// TwinCAT 3 PLC project SandBox
// ProgramVersion: 3.1.4026.22
// libraries:
//   [Logging Helper], * (Beckhoff Industrial)
//   Tc2_Standard, * (Beckhoff Automation GmbH)
//   Tc2_System, * (Beckhoff Automation GmbH)
// project tree:
//   / MAIN.TcPOU, PlcTask.TcTTO
//   Source/ MotionArgument.TcPOU, ST_MotionParameters.TcDUT
// (motion and I/O tree: see PLC project unittestplc)
// real-time tasks:
//   TASK PlcTask: cycle T#10ms, priority 20, ADS port 350
//   TASK PlcTask1: cycle T#10ms, priority 21, ADS port 351

CONFIGURATION SandBox
    RESOURCE PLC ON TwinCAT3
        TASK PlcTask(INTERVAL := T#10ms, PRIORITY := 21);
        PROGRAM MAIN WITH PlcTask : MAIN;
    END_RESOURCE
END_CONFIGURATION

// ---- Source/ST_MotionParameters.TcDUT
TYPE ST_MotionParameters :
	STRUCT
		Velocity : LREAL;
		Accel	 : LREAL;
		Decel	 : LREAL;
		Jerk	 : LREAL;
	END_STRUCT
END_TYPE

// ---- MAIN.TcPOU
PROGRAM MAIN
VAR
	Logger			: LogHelper<2>;
	LocalLog		: LocalLogger;
	initialized		: BOOL;
	Message			: LogMessage;
	Source			: LogSource;
	MotionArg		: MotionArgument;
	MotionParameters : ST_MotionParameters;
	
	//Commands
	logNoArgument	: BOOL;
	logWithArgument : BOOL;
END_VAR

IF NOT initialized THEN
	initialized			 := TRUE;
	MotionArg.Parameters REF= MotionParameters;
	Logger.Subscribe(LocalLog);
END_IF

IF logNoArgument THEN
	Source.SourceName := 'Test';
	Source.Timestamp := 123456789;
	Message.Message := 'Message';
	Message.Severity := 12;
	Logger.LogMessage(Source, Message);
	logNoArgument := FALSE;
END_IF

IF logWithArgument THEN
	Logger.LogMessage(Source, Message, MotionArg);
	logWithArgument := FALSE;
END_IF

END_PROGRAM

// ---- Source/MotionArgument.TcPOU
FUNCTION_BLOCK MotionArgument IMPLEMENTS I_LogArgument
VAR
	_Pars : REFERENCE TO ST_MotionParameters;
END_VAR

PROPERTY Parameters : REFERENCE TO ST_MotionParameters
GET
Parameters := _Pars;
END_GET
SET
_Pars REF= Parameters;
END_SET
END_PROPERTY

METHOD ToString : Logging_Helper.T_MaxString
ToString := CONCAT('Vel: ', CONCAT(TO_STRING(_Pars.Velocity), CONCAT(' Accel: ', CONCAT(TO_STRING(_Pars.Accel), CONCAT(' Decel: ', CONCAT(TO_STRING(_Pars.Decel), CONCAT(' Jerk: ',TO_STRING(_Pars.Jerk))))))));
END_METHOD

END_FUNCTION_BLOCK
